{attribute 'GeneratedUsingTerminal: EK1122-0000-0018'}
{attribute addProperty BoxType "EK1122-0000-0018"}
{attribute addProperty Id "Beckhoff_EL29xxsub_EK1100EK1100_AB5A94672"}
{attribute addProperty CRC "528969051"}
{attribute addProperty Size "2"}
TYPE Beckhoff_EL29xxEK1122_1F876D5B EXTENDS EK1122_AB5A9467 :
STRUCT
	{attribute addProperty Name "Beckhoff_EL29xxsub_EK1100"}
	Beckhoff_EL29xxsub_EK1100 : EK1100_AB5A9467;
END_STRUCT
END_TYPE

(* stored: Version 1.2.0.0, ProductVersion 3.1.4024.9
   DUT Beckhoff_EL29xxEK1122_1F876D5B: Id {1cbf7e91-c0ac-4dda-bba8-d2f34c6a7193} *)
